TYPE "UDT_ZC_COM_INT"
VERSION : 0.1
   STRUCT
      In : Int;
      Out : Int;
      Forzar : Bool;   // 0= Automatico / 1= Forzado
      ValorForzado : Int;   // Valor forzado
   END_STRUCT;

END_TYPE

